{attribute 'linkalways'} 
{attribute 'no_explicit_call' := 'This FB is a CLASS and must be accessed using methods or properties'}
{attribute 'enable_dynamic_creation'}
FUNCTION_BLOCK _TcVnArray10_ITcVnImage EXTENDS AliasDatatypeBase
VAR
	localData : TcVnArray10_ITcVnImage;
	activeData : REFERENCE TO TcVnArray10_ITcVnImage REF= localData;
	aliasBaseDatatype : _Array0to9OfITcVnImage;
END_VAR

PROPERTY PUBLIC Address : PVOID
GET
Address := ADR(activeData);
END_GET
END_PROPERTY

METHOD PUBLIC ClearReference
VAR_INPUT
END_VAR
activeData REF= localData;
SetBaseDatatypeReference();
END_METHOD

METHOD PUBLIC Clone : I_Datatype
VAR
    pClone : POINTER TO _TcVnArray10_ITcVnImage;
END_VAR
pClone := __NEW(_TcVnArray10_ITcVnImage);
Clone := pClone^;
END_METHOD

METHOD FB_init : BOOL
VAR_INPUT
	bInitRetains : BOOL; // if TRUE, the retain variables are initialized (warm start / cold start)
	bInCopyCode : BOOL;  // if TRUE, the instance afterwards gets moved into the copy code (online change)
	//InitialValue : TcVnArray10_ITcVnImage; // if possible, not all values can be initialized
END_VAR
//localData := InitialValue; // if possible, not all values can be initialized
SetBaseDatatypeReference();
AddBaseDatatype(aliasBaseDatatype);
END_METHOD

PROPERTY PUBLIC Identifier : T_MAXSTRING
GET
Identifier := 'TcVnArray10_ITcVnImage';
END_GET
END_PROPERTY

METHOD PUBLIC MakeReferenceTo
VAR_INPUT
	ReferenceTarget : REFERENCE TO TcVnArray10_ITcVnImage;
END_VAR
activeData REF= ReferenceTarget;
SetBaseDatatypeReference();
END_METHOD

METHOD PROTECTED SetBaseDatatypeReference
VAR_INPUT
END_VAR
aliasBaseDatatype.MakeReferenceTo(activeData);
END_METHOD

PROPERTY PUBLIC Size : UDINT
GET
Size := SIZEOF(activeData);
END_GET
END_PROPERTY

METHOD TryMakeReferenceTo : BOOL
VAR_INPUT
	Target : I_Datatype;
END_VAR
VAR
	targetAsAlias : I_AliasDatatype;
	pTargetData : POINTER TO TcVnArray10_ITcVnImage;
END_VAR
IF NOT Target.TryResolveAsAliasDatatype(targetAsAlias) THEN
	RETURN;
END_IF

IF targetAsAlias.Identifier <> Identifier THEN
	RETURN;
END_IF

pTargetData := Target.Address;
activeData REF= pTargetData^;
SetBaseDatatypeReference();
TryMakeReferenceTo := TRUE;
END_METHOD

PROPERTY PUBLIC Value : REFERENCE TO TcVnArray10_ITcVnImage
GET
Value REF= activeData;
END_GET
END_PROPERTY

END_FUNCTION_BLOCK

(* stored: Version 1.1.0.1, ProductVersion 3.1.4024.13
   POU _TcVnArray10_ITcVnImage: Id {d21ed5ae-434e-0398-1d34-d78e0e22bb0b}, SpecialFunc None
   Folder Core: Id {6c1db99e-bf7a-0bb3-088a-bea4354cec64}
   Folder Protected: Id {de5b51e7-46a9-06ab-2c36-30abe0b2442d}
   Folder Customize: Id {9440d840-7805-0f6a-337c-11d1f54ef919}
   Folder Constructor: Id {20b35323-f309-07fb-2fba-3a4a59a07bb7}
   Property Address: Id {2715513e-bb30-0807-3c76-cc0f72fd9291}
   Get Get: Id {5584efb0-78b8-0cd2-2c08-5da8eaa2854b}
   Method ClearReference: Id {994ffe60-bfbc-0b60-3451-772c89d828e9}
   Method Clone: Id {4f324a2d-a0f5-053a-1c81-a61883bb571a}
   Method FB_init: Id {1570272f-e78e-080d-0185-27ef69db7ed1}
   Property Identifier: Id {fd77efd1-6f6d-0543-00cc-60f18f0cd92a}
   Get Get: Id {1580796b-5810-0c17-33b8-f05a5d259ddc}
   Method MakeReferenceTo: Id {05f83d8c-d0e4-00f7-1237-4f9ab8aa6a5e}
   Method SetBaseDatatypeReference: Id {d6f66f45-b3d5-0cf9-0554-a3bff049d048}
   Property Size: Id {78383e4e-fb94-0b36-201a-7b9b43d70eda}
   Get Get: Id {e185d157-3c86-0b20-095b-a146bca4afc1}
   Method TryMakeReferenceTo: Id {46ce673d-4a3d-0473-332d-d093b56e6f94}
   Property Value: Id {9e03f9fb-8da5-0be9-248e-0adcb4700ed4}
   Get Get: Id {a278d222-85f4-0325-366f-97f785f9610b} *)
